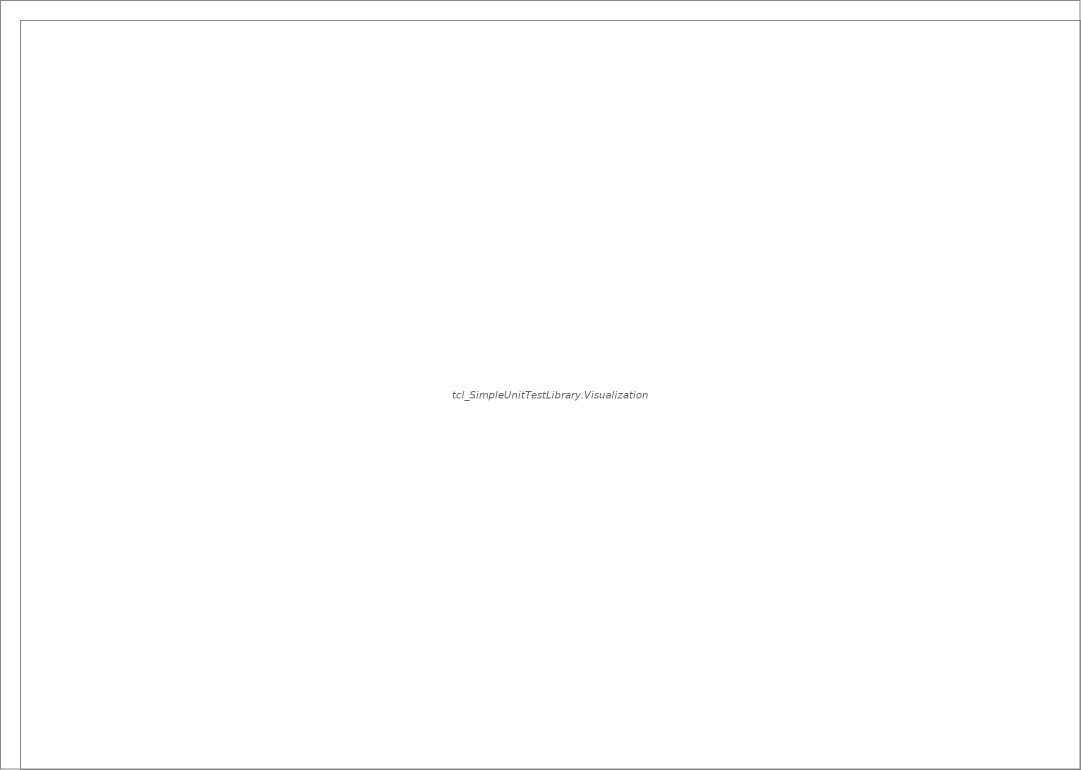
VISUALIZATION Visualization  // 1081x770
    Frame (20,20 1061x750)
        shows tcl_SimpleUnitTestLibrary.Visualization(TestRunner := PB_TestRunner.TestRunner, AssertionMessages := PB_TestRunner.TestRunner.AssertionMessages)
END_VISUALIZATION

(* stored: Version 1.1.0.1, ProductVersion 3.1.4024.6
   Visu Visualization: Id {ab61463a-dcf7-052a-1d55-6fd5b4702d10} *)
